FUNCTION_BLOCK GreenMasterSmokeControl extends GreenMasterSmokeControl_Base
VAR_INPUT
	{attribute 'TcEncoding':='UTF-8'}
	ModbusTCP_IP: STRING := '10.133.0.23';
	Exercise: BOOL;
	ResetSmokeDetectors: bool;
END_VAR
VAR_OUTPUT
	Exercising: BOOL;
	DamperError: BOOL;
END_VAR
VAR
	ModbusTCP: ModbusTCP;
	DamperControl: DamperControl;
	DamperModule_0: DamperModule;
	DamperModule_1: DamperModule;
	DamperModule_2: DamperModule;
	DamperModule_3: DamperModule;
	DamperModule_4: DamperModule;
	DamperModule_5: DamperModule;
	DamperModule_6: DamperModule;
	DamperModule_7: DamperModule;
	DamperModule_8: DamperModule;
	DamperModule_9: DamperModule;
	DamperModule_10: DamperModule;
	DamperModule_11: DamperModule;
	DamperModule_12: DamperModule;
	DamperModule_13: DamperModule;
	DamperModule_14: DamperModule;
	DamperModule_15: DamperModule;
END_VAR


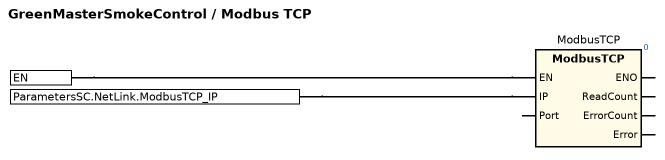
// PAGE Modbus TCP
ModbusTCP(EN := EN, IP := ParametersSC.NetLink.ModbusTCP_IP);

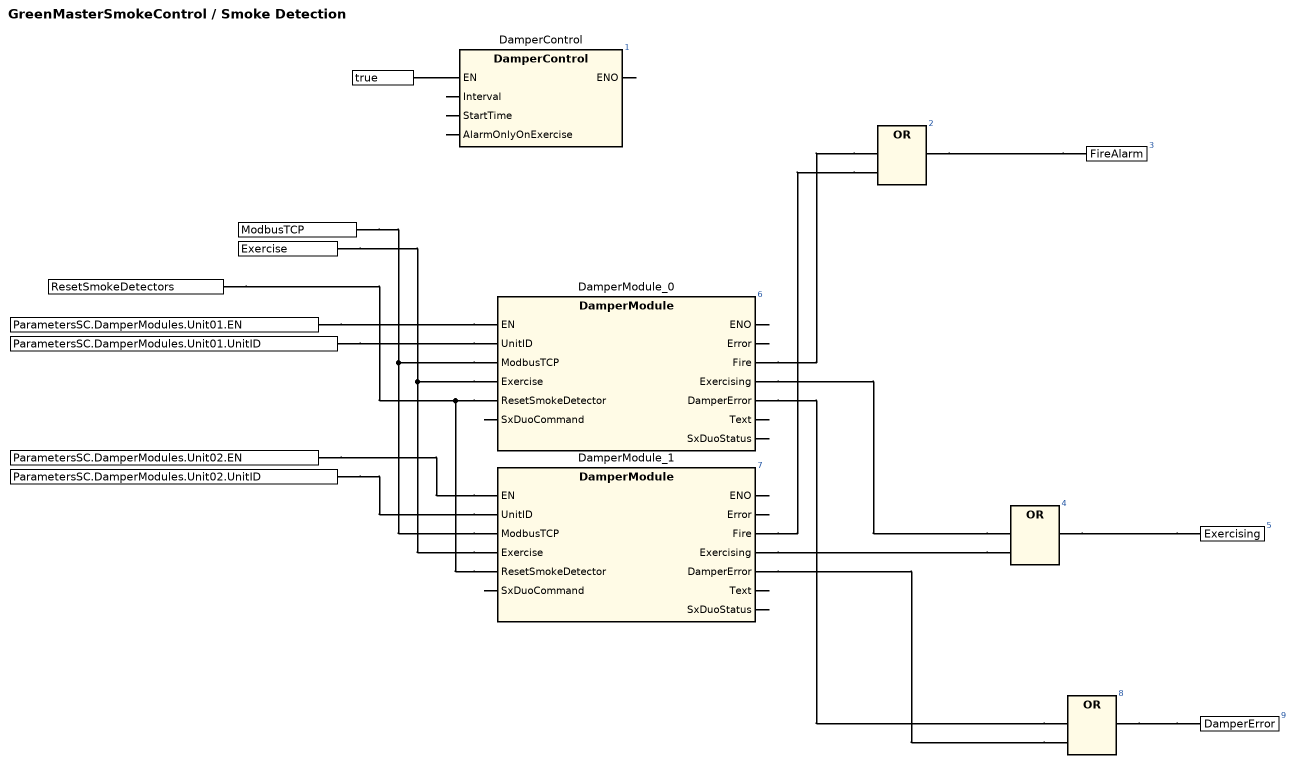
// PAGE Smoke Detection
DamperControl(EN := true);
FireAlarm := DamperModule_0.Fire OR DamperModule_1.Fire;
Exercising := DamperModule_0.Exercising OR DamperModule_1.Exercising;
DamperModule_0(
    EN := ParametersSC.DamperModules.Unit01.EN,
    UnitID := ParametersSC.DamperModules.Unit01.UnitID,
    ModbusTCP := ModbusTCP,
    Exercise := Exercise,
    ResetSmokeDetector := ResetSmokeDetectors); // DamperModule
DamperModule_1(
    EN := ParametersSC.DamperModules.Unit02.EN,
    UnitID := ParametersSC.DamperModules.Unit02.UnitID,
    ModbusTCP := ModbusTCP,
    Exercise := Exercise,
    ResetSmokeDetector := ResetSmokeDetectors); // DamperModule
DamperError := DamperModule_0.DamperError OR DamperModule_1.DamperError;

METHOD Update : BOOL
VAR_INPUT
	Parameters: REFERENCE TO GreenMasterBaseParameters;
	ParametersSC: REFERENCE TO SmokeControlParametersBase;
END_VAR
VAR
	TempAlarm: bool;
END_VAR
ParametersSC.DamperModules.Unit01.Update(Parameters, DamperModule_0);
ParametersSC.DamperModules.Unit02.Update(Parameters, DamperModule_1);
ParametersSC.DamperModules.Unit03.Update(Parameters, DamperModule_3);
ParametersSC.DamperModules.Unit04.Update(Parameters, DamperModule_4);
ParametersSC.DamperModules.Unit05.Update(Parameters, DamperModule_5);
ParametersSC.DamperModules.Unit06.Update(Parameters, DamperModule_6);
ParametersSC.DamperModules.Unit07.Update(Parameters, DamperModule_7);
ParametersSC.DamperModules.Unit08.Update(Parameters, DamperModule_8);
ParametersSC.DamperModules.Unit09.Update(Parameters, DamperModule_9);
ParametersSC.DamperModules.Unit10.Update(Parameters, DamperModule_10);
ParametersSC.DamperModules.Unit11.Update(Parameters, DamperModule_11);
ParametersSC.DamperModules.Unit12.Update(Parameters, DamperModule_12);
ParametersSC.DamperModules.Unit13.Update(Parameters, DamperModule_13);
ParametersSC.DamperModules.Unit14.Update(Parameters, DamperModule_14);
ParametersSC.DamperModules.Unit15.Update(Parameters, DamperModule_15);


Parameters.Alarm.Status.A.FireExtractExternal := 
	(ParametersSC.DamperModules.Unit01.Fire AND ParametersSC.DamperModules.Unit01.CentralFireAlarm) OR
	(ParametersSC.DamperModules.Unit02.Fire AND ParametersSC.DamperModules.Unit02.CentralFireAlarm) OR
	(ParametersSC.DamperModules.Unit03.Fire AND ParametersSC.DamperModules.Unit03.CentralFireAlarm) OR
	(ParametersSC.DamperModules.Unit04.Fire AND ParametersSC.DamperModules.Unit04.CentralFireAlarm) OR
	(ParametersSC.DamperModules.Unit05.Fire AND ParametersSC.DamperModules.Unit05.CentralFireAlarm) OR
	(ParametersSC.DamperModules.Unit06.Fire AND ParametersSC.DamperModules.Unit06.CentralFireAlarm) OR
	(ParametersSC.DamperModules.Unit07.Fire AND ParametersSC.DamperModules.Unit07.CentralFireAlarm) OR
	(ParametersSC.DamperModules.Unit08.Fire AND ParametersSC.DamperModules.Unit08.CentralFireAlarm) OR
	(ParametersSC.DamperModules.Unit09.Fire AND ParametersSC.DamperModules.Unit09.CentralFireAlarm) OR
	(ParametersSC.DamperModules.Unit10.Fire AND ParametersSC.DamperModules.Unit10.CentralFireAlarm) OR
	(ParametersSC.DamperModules.Unit11.Fire AND ParametersSC.DamperModules.Unit11.CentralFireAlarm) OR
	(ParametersSC.DamperModules.Unit12.Fire AND ParametersSC.DamperModules.Unit12.CentralFireAlarm) OR
	(ParametersSC.DamperModules.Unit13.Fire AND ParametersSC.DamperModules.Unit13.CentralFireAlarm) OR
	(ParametersSC.DamperModules.Unit14.Fire AND ParametersSC.DamperModules.Unit14.CentralFireAlarm) OR
	(ParametersSC.DamperModules.Unit15.Fire AND ParametersSC.DamperModules.Unit15.CentralFireAlarm);
	
Parameters.Alarm.Status.A.FireLocal := 
	(ParametersSC.DamperModules.Unit01.Fire AND NOT ParametersSC.DamperModules.Unit01.CentralFireAlarm) OR
	(ParametersSC.DamperModules.Unit02.Fire AND NOT ParametersSC.DamperModules.Unit02.CentralFireAlarm) OR
	(ParametersSC.DamperModules.Unit03.Fire AND NOT ParametersSC.DamperModules.Unit03.CentralFireAlarm) OR
	(ParametersSC.DamperModules.Unit04.Fire AND NOT ParametersSC.DamperModules.Unit04.CentralFireAlarm) OR
	(ParametersSC.DamperModules.Unit05.Fire AND NOT ParametersSC.DamperModules.Unit05.CentralFireAlarm) OR
	(ParametersSC.DamperModules.Unit06.Fire AND NOT ParametersSC.DamperModules.Unit06.CentralFireAlarm) OR
	(ParametersSC.DamperModules.Unit07.Fire AND NOT ParametersSC.DamperModules.Unit07.CentralFireAlarm) OR
	(ParametersSC.DamperModules.Unit08.Fire AND NOT ParametersSC.DamperModules.Unit08.CentralFireAlarm) OR
	(ParametersSC.DamperModules.Unit09.Fire AND NOT ParametersSC.DamperModules.Unit09.CentralFireAlarm) OR
	(ParametersSC.DamperModules.Unit10.Fire AND NOT ParametersSC.DamperModules.Unit10.CentralFireAlarm) OR
	(ParametersSC.DamperModules.Unit11.Fire AND NOT ParametersSC.DamperModules.Unit11.CentralFireAlarm) OR
	(ParametersSC.DamperModules.Unit12.Fire AND NOT ParametersSC.DamperModules.Unit12.CentralFireAlarm) OR
	(ParametersSC.DamperModules.Unit13.Fire AND NOT ParametersSC.DamperModules.Unit13.CentralFireAlarm) OR
	(ParametersSC.DamperModules.Unit14.Fire AND NOT ParametersSC.DamperModules.Unit14.CentralFireAlarm) OR
	(ParametersSC.DamperModules.Unit15.Fire AND NOT ParametersSC.DamperModules.Unit15.CentralFireAlarm);
END_METHOD

METHOD Write : BOOL
VAR_INPUT
END_VAR
DamperModule_0.StartWrite();
DamperModule_1.StartWrite();
END_METHOD

END_FUNCTION_BLOCK

(* stored: Version 1.1.0.1, ProductVersion 3.1.4024.6
   POU GreenMasterSmokeControl: Id {be7d3d16-f182-463d-92da-aec7fbfb4c74}, SpecialFunc None
   Method Update: Id {ab80fefc-edf0-479d-a8ce-d6df8d540431}
   Method Write: Id {71f1c73f-c6fa-4914-b408-5a220d42ac75} *)
